// SIMATIC S7-200 project (STEP 7-Micro/WIN), CPU 221 REL 01.10

ORGANIZATION_BLOCK MAIN:OB1
TITLE=PROGRAM COMMENTS
BEGIN
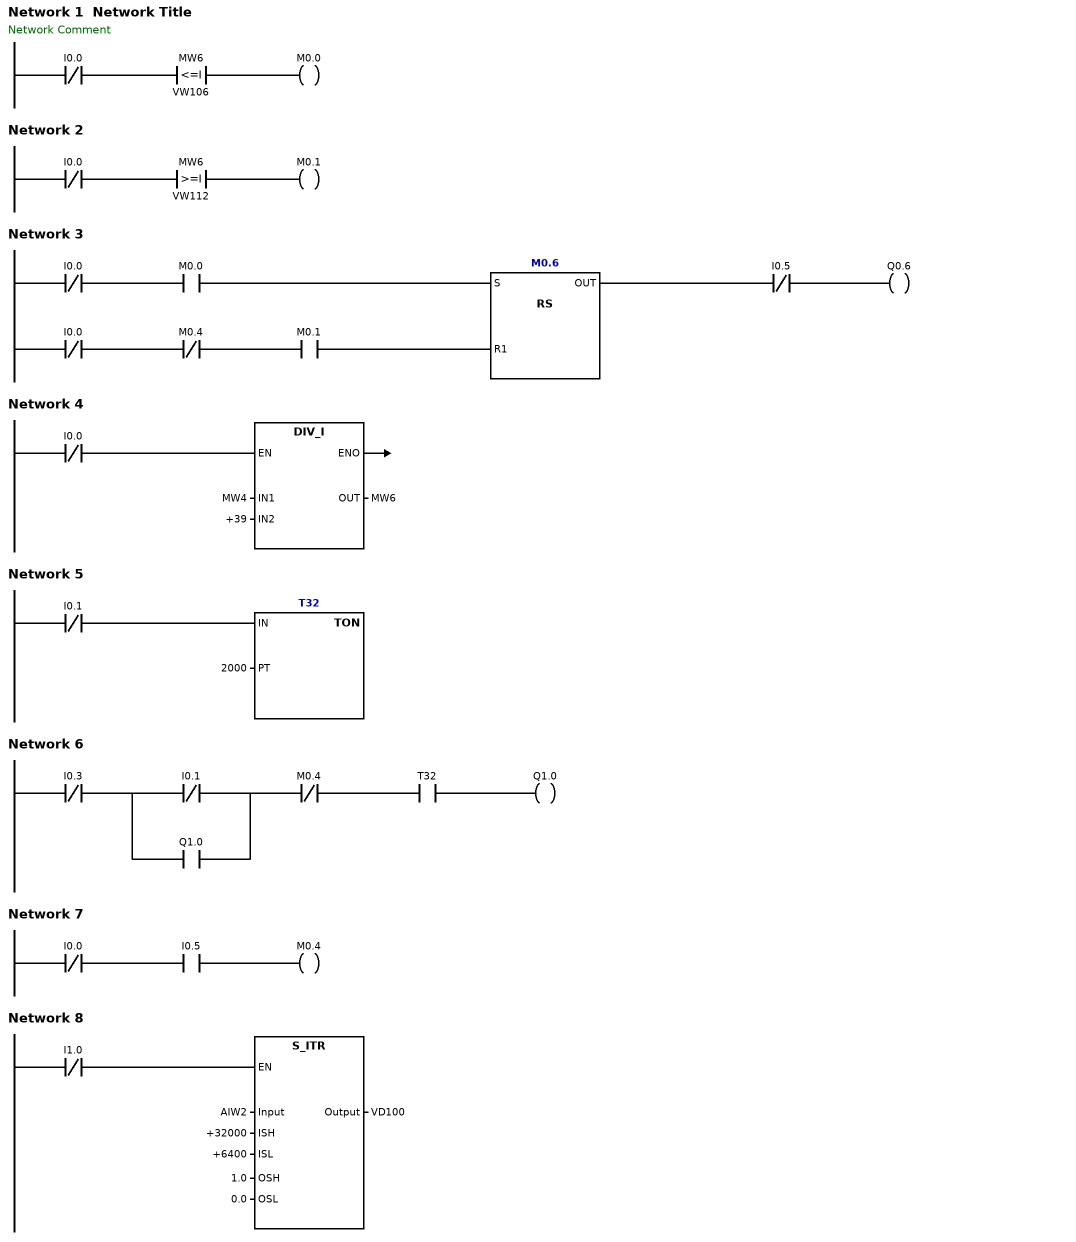
Network 1 // Network Title
// Network Comment
LDN    I0.0
AW<=   MW6, VW106
=      M0.0
Network 2
LDN    I0.0
AW>=   MW6, VW112
=      M0.1
Network 3
LDN    I0.0
A      M0.0
LDN    I0.0
AN     M0.4
A      M0.1
NOT
LPS
A      M0.6
=      M0.6
LPP
ALD
O      M0.6
=      M0.6
AN     I0.5
=      Q0.6
Network 4
LDN    I0.0
MOVW   MW4, MW6
/I     +39, MW6
Network 5
LDN    I0.1
TON    T32, 2000
Network 6
LDN    I0.3
LDN    I0.1
O      Q1.0
ALD
AN     M0.4
A      T32
=      Q1.0
Network 7
LDN    I0.0
A      I0.5
=      M0.4
Network 8
LDN    I1.0
CALL   S_ITR:SBR1, AIW2, +32000, +6400, 1.0, 0.0, VD100
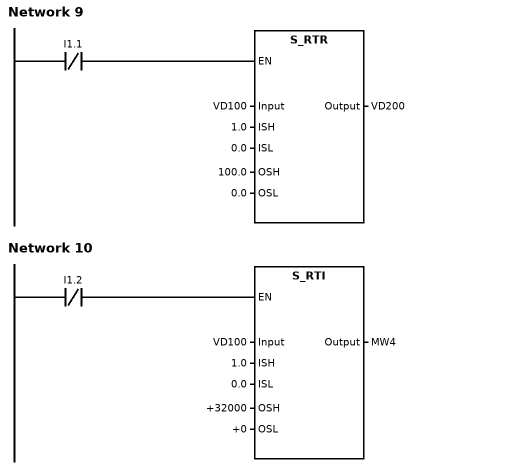
Network 9
LDN    I1.1
CALL   S_RTR:SBR2, VD100, 1.0, 0.0, 100.0, 0.0, VD200
Network 10
LDN    I1.2
CALL   S_RTI:SBR3, VD100, 1.0, 0.0, +32000, +0, MW4
END_ORGANIZATION_BLOCK

SUBROUTINE_BLOCK SBR_0:SBR0
TITLE=SUBROUTINE COMMENTS
BEGIN
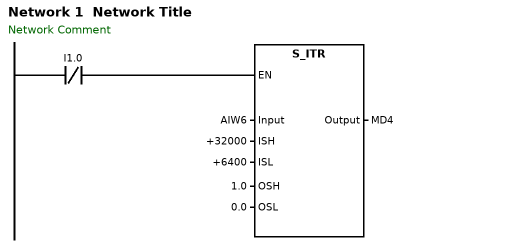
Network 1 // Network Title
// Network Comment
LDN    I1.0
CALL   S_ITR:SBR1, AIW6, +32000, +6400, 1.0, 0.0, MD4
END_SUBROUTINE_BLOCK

// SBR1: protected block, not included

// SBR2: protected block, not included

// SBR3: protected block, not included
